// TIA Portal V20 export
TYPE "UDT_typePosCtrl"
   STRUCT
      input : Struct
         bo_estop : Bool;
         bo_enable : Bool;
         bo_reset : Bool;
         bo_home : Bool;
         bo_jogforward : Bool;
         bo_jogbackward : Bool;
         bo_movevelocity : Bool;
         bo_posabsolute : Bool;
         bo_posrelative : Bool;
         bo_gearin : Bool;
         bo_camin : Bool;
         bo_camout : Bool;
         bo_halt : Bool;
         bo_stop : Bool;
         configuration : Struct
            home { ExternalWritable := 'False'} : Struct
               i16_mode : Int;
               r64_homeposition : LReal;
               r64_ApproachVelocity : LReal := 10.0;
               r64_ReferencingVelocity : LReal := 5.0;
            END_STRUCT;
            jog : Struct
               r64_velocity : LReal := 5.0;
               r64_acceleration : LReal := 1000.0;
               r64_jerk : LReal := -1.0;
            END_STRUCT;
            movevelocity : Struct
               r64_velocity : LReal := 10.0;
               r64_acceleration : LReal := 1000.0;
               r64_jerk : LReal := -1.0;
               i16_direction : Int;
            END_STRUCT;
            posabsolute : Struct
               r64_velocity : LReal := 10.0;
               r64_position : LReal := 0.0;
               r64_acceleration : LReal := 1000.0;
               r64_jerk : LReal := -1.0;
               i16_direction : Int := 1;
            END_STRUCT;
            posrelative : Struct
               r64_velocity : LReal := 10.0;
               r64_position : LReal := 0.0;
               r64_acceleration : LReal := 1000.0;
               r64_jerk : LReal := -1.0;
            END_STRUCT;
            gearin : Struct
               RatioNumerator : DInt := 1;
               RatioDenominator : DInt := 1;
            END_STRUCT;
            camin : Struct
               i16_syncProfileReference : Int := 2;
               i16_applicationMode : Int := 0;
               r64_masterStartDistance : LReal;
               r64_masterSyncPosition : LReal;
               r64_masterOffset : LReal;
            END_STRUCT;
         END_STRUCT;
      END_STRUCT;
      output : Struct
         bo_communicationOk : Bool;
         bo_enabled : Bool;
         bo_homed : Bool;
         bo_inGear : Bool;
         bo_StarSync : Bool;
         bo_inSync : Bool;
         bo_fault : Bool;
         bo_endprofile : Bool;
         bo_SWLimitMinActived : Bool;
         bo_SWLimitMaxActived : Bool;
         bo_HWLimitMinActived : Bool;
         bo_HWLimitMaxActived : Bool;
         r64_actualVelocity : LReal;
         r64_actualPosition : LReal;
      END_STRUCT;
   END_STRUCT;
END_TYPE
